// TwinCAT 3 PLC project PLC
// ProgramVersion: 3.1.4024.0
// libraries:
//   Tc2_Standard, * (Beckhoff Automation GmbH)
//   Tc2_System, * (Beckhoff Automation GmbH)
//   Tc3_Module, * (Beckhoff Automation GmbH)
// project tree:
//   GVLs/ GVL_Kitchen.TcGVL
//   / PlcTask.TcTTO, Task_Cutter.TcTTO
//   POUs/ MAIN_Burner.TcPOU, MAIN_Cutter.TcPOU
// real-time tasks:
//   TASK Task Burner: cycle T#10ms, priority 20, ADS port 350
//   TASK Task Cutter: cycle T#10ms, priority 21, ADS port 352
//   TASK Delay: cycle T#10ms, priority 1, ADS port 351

CONFIGURATION PLC
    RESOURCE PLC ON TwinCAT3
        TASK PlcTask(INTERVAL := T#10ms, PRIORITY := 20);
        TASK Task_Cutter(INTERVAL := T#10ms, PRIORITY := 21);
        PROGRAM MAIN_Burner WITH PlcTask : MAIN_Burner;
        PROGRAM MAIN_Cutter WITH Task_Cutter : MAIN_Cutter;
    END_RESOURCE
END_CONFIGURATION

// ---- GVLs/GVL_Kitchen.TcGVL
{attribute 'qualified_only'}
VAR_GLOBAL
	
	System_Start : Int := 1;
	Food_Cut	 : INT  := 0;
	Food_Spiced  : INT  := 0;
	Food_Cooked  : INT  := 0;
	Food_Plated  : INT  := 0;
END_VAR

// ---- POUs/MAIN_Burner.TcPOU
PROGRAM MAIN_Burner
VAR

	Delay: TON;
	IN: BOOL;
	PT: TIME;
	Q: INT;
	State : Int;
END_VAR

IF GVL_Kitchen.System_Start = 0 THEN
 	 	
					Delay(IN:=TRUE, PT:=T#1S);
					IF NOT(Delay.Q) THEN
					   RETURN;
					END_IF
					Delay(IN:=FALSE);
					
ELSE	
		CASE State OF
		0: 
		IF GVL_kitchen.Food_Spiced >0 THEN
			
			 		Delay(IN:=TRUE, PT:=T#7S);
					IF NOT(Delay.Q) THEN
					   RETURN;
					END_IF
					Delay(IN:=FALSE);
			
			GVL_kitchen.Food_Spiced := GVL_kitchen.Food_Spiced-1;
			GVL_Kitchen.Food_Cooked := GVL_Kitchen.Food_Cooked +1;
			State := 1;
			END_IF;
			
		1: 
		IF GVL_kitchen.Food_cooked > 0 THEN
				 	
					Delay(IN:=TRUE, PT:=T#3S);
					IF NOT(Delay.Q) THEN
					   RETURN;
					END_IF
					Delay(IN:=FALSE);
					
			GVL_Kitchen.Food_Cooked := GVL_Kitchen.Food_Cooked -1;
			GVL_Kitchen.Food_Plated := GVL_Kitchen.Food_Plated +1;
			ELSE 
				state := 0;
			END_IF;
		END_CASE 
END_IF

END_PROGRAM

// ---- POUs/MAIN_Cutter.TcPOU
PROGRAM MAIN_Cutter
VAR

	Delay: TON;
	IN: BOOL;
	PT: TIME;
	Q: INT;
	State : INT;
END_VAR

IF GVL_Kitchen.System_Start = 0 THEN
 		Delay(IN:=TRUE, PT:=T#1S);
		IF NOT(Delay.Q) THEN
		   RETURN;
		END_IF
		Delay(IN:=FALSE);
	ELSE	
		CASE State OF
		0: 
			IF GVL_kitchen.Food_Cut < 2 THEN
				
					Delay(IN:=TRUE, PT:=T#5S);
					IF NOT(Delay.Q) THEN
					   RETURN;
					END_IF
					Delay(IN:=FALSE);
				
				GVL_Kitchen.Food_Cut := GVL_Kitchen.Food_Cut +1;
				ELSE 
					state := 1;
			END_IF;
		1:
			IF GVL_kitchen.Food_Spiced < 2 THEN
			 		
					Delay(IN:=TRUE, PT:=T#3S);
					IF NOT(Delay.Q) THEN
					   RETURN;
					END_IF
					Delay(IN:=FALSE);
					
				GVL_Kitchen.Food_Cut := GVL_Kitchen.Food_Cut -1;
				GVL_Kitchen.Food_Spiced := GVL_Kitchen.Food_Spiced +1;
				ELSE
				state := 0;
			END_IF;
		
		
		END_CASE
END_IF

END_PROGRAM
